(* IEC 61131-3 sources: Industry-PLC-LLM/data/PLCBEAD_repo/PLCBEAD_PLCEmbed-main/PLC-BEAD/Source/GEB/COUNT_BR, 1 file *)

(* ---- COUNT_BR.ST ---- *)
FUNCTION _BYTE_TO_INT:INT
	VAR_INPUT
		IN :	BYTE;
	END_VAR

	_BYTE_TO_INT := USINT_TO_INT(BYTE_TO_USINT(IN));

END_FUNCTION

FUNCTION INC:INT
	VAR_INPUT
		X :	INT;
		D :	INT;
		M :	INT;
	END_VAR

	INC := (X + D + M + 1) MOD (M + 1);
END_FUNCTION

FUNCTION_BLOCK COUNT_BR
	VAR_INPUT
		SET :	BOOL;
		IN :	BYTE;
		UP :	BOOL;
		DN :	BOOL;
		STEPP :	BYTE := BYTE#1;
		MX :	BYTE := BYTE#255;
		RST :	BOOL;
	END_VAR
	VAR_OUTPUT
		CNT :	BYTE;
	END_VAR

	VAR
		last_up :	BOOL;
		last_dn :	BOOL;
	END_VAR

	IF RST THEN
		CNT := BYTE#0;
	ELSIF SET THEN
		CNT := INT_TO_BYTE(LIMIT(0,_BYTE_TO_INT(IN),_BYTE_TO_INT(MX)));
	ELSIF UP AND NOT last_up THEN
		CNT := INT_TO_BYTE(INC(_BYTE_TO_INT(CNT),_BYTE_TO_INT(STEPP),_BYTE_TO_INT(MX)));
	ELSIF DN AND NOT last_dn THEN
		CNT := INT_TO_BYTE(INC(_BYTE_TO_INT(CNT),_BYTE_TO_INT(STEPP) * -1,_BYTE_TO_INT(MX)));
	END_IF;
	last_up := UP;
	last_dn := DN;
END_FUNCTION_BLOCK

PROGRAM program0
  VAR
	SET :	BOOL;
	IN :	BYTE;
	UP :	BOOL;
	DN :	BOOL;
	STEPP:	BYTE;
	MX :	BYTE;
	RST :	BOOL;

	CNT :	BYTE;
	func_block : COUNT_BR;
  END_VAR
	func_block.SET  :=SET  ;
	func_block.IN   :=IN   ;
	func_block.UP   :=UP   ;
	func_block.DN   :=DN   ;
	func_block.STEPP :=STEPP ;
	func_block.MX   :=MX   ;
	func_block.RST  :=RST  ;

	func_block();
	CNT := func_block.CNT;
END_PROGRAM
